{attribute 'linkalways'} 
{attribute 'no_explicit_call' := 'This FB is a CLASS and must be accessed using methods or properties'}
{attribute 'enable_dynamic_creation'}
FUNCTION_BLOCK _LREAL EXTENDS NumericDatatypeBase
VAR
	localData : LREAL;
	activeData : REFERENCE TO LREAL REF= localData;
END_VAR

PROPERTY PUBLIC Address : PVOID
GET
Address := ADR(activeData);
END_GET
END_PROPERTY

METHOD PUBLIC ClearReference
VAR_INPUT
END_VAR
activeData REF= localData;
END_METHOD

METHOD PUBLIC Clone : I_Datatype
VAR
    pClone : POINTER TO _LREAL;
END_VAR
pClone := __NEW(_LREAL(InitialValue := Value));
Clone := pClone^;
END_METHOD

METHOD FB_init : BOOL
VAR_INPUT
	bInitRetains : BOOL; // if TRUE, the retain variables are initialized (warm start / cold start)
	bInCopyCode : BOOL;  // if TRUE, the instance afterwards gets moved into the copy code (online change)
	InitialValue : LREAL;
END_VAR
localData := InitialValue;
END_METHOD

PROPERTY PUBLIC IsFloat : BOOL
GET
IsFloat := TRUE;
END_GET
END_PROPERTY

PROPERTY PUBLIC IsSigned : BOOL
GET
IsSigned := TRUE;
END_GET
END_PROPERTY

METHOD PUBLIC MakeReferenceTo
VAR_INPUT
	ReferenceTarget : REFERENCE TO LREAL;
END_VAR
activeData REF= ReferenceTarget;
END_METHOD

PROPERTY PUBLIC MaxValue : LREAL
GET
MaxValue :=  DatatypeLimits.LREAL_MAX_VALUE;
END_GET
END_PROPERTY

PROPERTY PUBLIC MinValue : LREAL
GET
MinValue := DatatypeLimits.LREAL_MIN_VALUE;
END_GET
END_PROPERTY

METHOD PROTECTED SerializeMaxValue
VAR_INPUT
	Serializer : I_Serializer;
END_VAR
Serializer.AddLreal(MaxValue);
END_METHOD

METHOD PROTECTED SerializeMinValue
VAR_INPUT
	Serializer : I_Serializer;
END_VAR
Serializer.AddLreal(MinValue);
END_METHOD

METHOD PUBLIC SerializeWith
VAR_INPUT
	Serializer : I_Serializer;
END_VAR
Serializer.AddLreal(activeData);
END_METHOD

PROPERTY PUBLIC Size : UDINT
GET
Size := SIZEOF(activeData);
END_GET
END_PROPERTY

METHOD TryDeserializeFrom : BOOL
VAR_INPUT
	Deserializer : I_Deserializer;
	Feedback : I_DeserializerFeedback;
END_VAR
TryDeserializeFrom := Deserializer.TryGetLreal(activeData, Feedback);
END_METHOD

METHOD TryMakeReferenceTo : BOOL
VAR_INPUT
	Target : I_Datatype;
END_VAR
VAR
	pTargetData : POINTER TO LREAL;
END_VAR
IF NOT (Target.TypeName = TypeName) THEN
	RETURN;
END_IF

pTargetData := Target.Address;
activeData REF= pTargetData^;
TryMakeReferenceTo := TRUE;
END_METHOD

PROPERTY PUBLIC TypeName : T_MAXSTRING
GET
TypeName := 'LREAL';
END_GET
END_PROPERTY

PROPERTY PUBLIC Value : REFERENCE TO LREAL
GET
Value REF= activeData;
END_GET
END_PROPERTY

END_FUNCTION_BLOCK

(* stored: Version 1.1.0.1, ProductVersion 3.1.4024.12
   POU _LREAL: Id {6481f43c-f724-4fdc-8169-15211a7421ae}, SpecialFunc None
   Folder Constructor: Id {01b0dc38-39ba-4b04-a774-579f98db0c8a}
   Folder Protected: Id {d6c987bd-bc52-06e0-1426-68be4cd615ca}
   Property Address: Id {64846ad0-ecd1-4bc1-8c14-0ae1c4a8facb}
   Get Get: Id {5c1e99a4-dd80-4e12-b0e5-7204dbf767f3}
   Method ClearReference: Id {2cbe2f04-1c1f-4c5e-b15b-afad6184c509}
   Method Clone: Id {5d0e0753-7aa1-48a4-96f2-2dcc6aec1ea8}
   Method FB_init: Id {5948e398-3883-4c50-844e-9e60f4eebb06}
   Property IsFloat: Id {66555880-1394-414a-a3a9-a083b1297209}
   Get Get: Id {5e8cc673-116a-4024-b83a-96aeecf56f77}
   Property IsSigned: Id {446a64f6-bd45-4525-b735-b5996051aa99}
   Get Get: Id {2413006a-9bc9-4170-9612-5768f95f3e89}
   Method MakeReferenceTo: Id {655cc873-c33a-416b-b99d-1a30b2b10923}
   Property MaxValue: Id {243f2af4-685e-0e25-07d5-f2dc2199d217}
   Get Get: Id {237997de-4e7e-02e3-319d-a83305687d18}
   Property MinValue: Id {dc91090d-486c-0029-2ff5-220e8e4e4305}
   Get Get: Id {7f1294b5-708a-0259-0a85-0991c18e2144}
   Method SerializeMaxValue: Id {ed114e15-c7c6-0c3f-2500-af86fb06a2cf}
   Method SerializeMinValue: Id {cd89fd53-18db-0cf8-3684-549fca515832}
   Method SerializeWith: Id {aa2ea405-4385-4112-8715-309123710b6b}
   Property Size: Id {214679cd-9001-4a6e-b59f-5128ca94fffc}
   Get Get: Id {f29c8af4-b7c3-4441-a0c3-39feb51051ae}
   Method TryDeserializeFrom: Id {9b98f558-5f87-4c6d-af16-5fc6a6173c5e}
   Method TryMakeReferenceTo: Id {46dd4ca3-00ca-41c7-80be-900b1eb0869f}
   Property TypeName: Id {0cb6ef98-c842-4fb9-9516-b4d8f991a80f}
   Get Get: Id {52ca1e18-c9a5-4cb3-b7a4-30c8caeefe7a}
   Property Value: Id {8f843798-4d8f-437c-8356-78b44d9e5022}
   Get Get: Id {7df50172-339b-4c76-98e1-713a7cc1aac6} *)
